// TwinCAT 3 PLC project Untitled1
// ProgramVersion: 3.1.4024.0
// libraries:
//   Tc2_Standard, * (Beckhoff Automation GmbH)
//   Tc2_System, * (Beckhoff Automation GmbH)
//   Tc3_Module, * (Beckhoff Automation GmbH)
// project tree:
//   / GlobalTextList.TcGTLO, PlcTask.TcTTO, Visualization Manager.TcVMO (not stored)
//   GVLs/ GIOL.TcGVL, Global_IO_assignment.TcPOU (not stored), GVL.TcGVL
//   POUs/ BINARY_TO_DEC.TcPOU, BLINK.TcPOU (not stored), MAIN.TcPOU, INMODE.TcPOU, Pulse.TcPOU, ROBOT_BIT_TRL.TcPOU
//   VISUs/ StandardPLCversenyVISU.TcVIS
// real-time tasks:
//   TASK PlcTask: cycle T#10ms, priority 20, ADS port 350
// I/O:
//   DEVICE Device 1 (EtherCAT), AmsNetId 5.86.98.224.2.1
//     Term 1 (EK1200) [EK1200-5000 EtherCAT Power supply (2A E-Bus)]
//       Term 2 (EL1008) [EL1008 8Ch. Dig. Input 24V, 3ms]
//       Term 3 (EL1008) [EL1008 8Ch. Dig. Input 24V, 3ms]
//       Term 4 (EL2008) [EL2008 8Ch. Dig. Output 24V, 0.5A]
//       Term 5 (EL2008) [EL2008 8Ch. Dig. Output 24V, 0.5A]
//       Term 6 (EL9011) [EL9011 End Terminal]
// variable links:
//   Untitled1/Untitled1 Instance <-> Device 1 (EtherCAT)/Term 1 (EK1200)/Term 2 (EL1008)
//     PlcTask Inputs/GIOL.xIn{0..7} <-> Channel {1..8}/Input  (8 links)
//   Untitled1/Untitled1 Instance <-> Device 1 (EtherCAT)/Term 1 (EK1200)/Term 3 (EL1008)
//     PlcTask Inputs/GIOL.xIn{8..15} <-> Channel {1..8}/Input  (8 links)
//   Untitled1/Untitled1 Instance <-> Device 1 (EtherCAT)/Term 1 (EK1200)/Term 4 (EL2008)
//     PlcTask Outputs/GIOL.Out{0..7} <-> Channel {1..8}/Output  (8 links)
//   Untitled1/Untitled1 Instance <-> Device 1 (EtherCAT)/Term 1 (EK1200)/Term 5 (EL2008)
//     PlcTask Outputs/GIOL.Out{8..15} <-> Channel {1..8}/Output  (8 links)

CONFIGURATION Untitled1
    RESOURCE PLC ON TwinCAT3
        TASK PlcTask(INTERVAL := T#10ms, PRIORITY := 20);
        PROGRAM MAIN WITH PlcTask : MAIN;
    END_RESOURCE
END_CONFIGURATION

// ---- GVLs/GIOL.TcGVL
{attribute 'qualified_only'}
VAR_GLOBAL
	xIn0 	AT%IX0.0:	BOOL;
	xIn1 	AT%IX0.1:	BOOL;
	xIn2 	AT%IX0.2:	BOOL;
	xIn3 	AT%IX0.3:	BOOL;
	xIn4 	AT%IX0.4:	BOOL;
	xIn5 	AT%IX0.5:	BOOL;
	xIn6 	AT%IX0.6:	BOOL;
	xIn7 	AT%IX0.7:	BOOL;
	
	xIn8 	AT%IX1.0:	BOOL;
	xIn9 	AT%IX1.1:	BOOL;
	xIn10 	AT%IX1.2:	BOOL;
	xIn11 	AT%IX1.3:	BOOL;
	xIn12 	AT%IX1.4:	BOOL;
	xIn13 	AT%IX1.5:	BOOL;
	xIn14 	AT%IX1.6:	BOOL;
	xIn15 	AT%IX1.7:	BOOL;
	
	Out0 	AT%QX0.0:	BOOL;
	Out1 	AT%QX0.1:	BOOL;
	Out2 	AT%QX0.2:	BOOL;
	Out3 	AT%QX0.3:	BOOL;
	Out4 	AT%QX0.4:	BOOL;
	Out5 	AT%QX0.5:	BOOL;
	Out6 	AT%QX0.6:	BOOL;
	Out7 	AT%QX0.7:	BOOL;
	
	
	Out8 	AT%QX1.0:	BOOL;
	Out9 	AT%QX1.1:	BOOL;
	Out10 	AT%QX1.2:	BOOL;
	Out11 	AT%QX1.3:	BOOL;
	Out12 	AT%QX1.4:	BOOL;
	Out13 	AT%QX1.5:	BOOL;
	Out14 	AT%QX1.6:	BOOL;
	Out15 	AT%QX1.7:	BOOL;
	
	In0 	:	BOOL;
	In1 	:	BOOL;
	In2 	:	BOOL;
	In3 	:	BOOL;
	In4 	:	BOOL;
	In5 	:	BOOL;
	In6 	:	BOOL;
	In7 	:	BOOL;
	
	In8 	:	BOOL;
	In9 	:	BOOL;
	In10 	:	BOOL;
	In11 	:	BOOL;
	In12 	:	BOOL;
	In13 	:	BOOL;
	In14 	:	BOOL;
	In15 	:	BOOL;
	
	bIn0 	:	BOOL;
	bIn1 	:	BOOL;
	bIn2 	:	BOOL;
	bIn3 	:	BOOL;
	bIn4 	:	BOOL;
	bIn5 	:	BOOL;
	bIn6 	:	BOOL;
	bIn7 	:	BOOL;
	
	bIn8 	:	BOOL;
	bIn9 	:	BOOL;
	bIn10 	:	BOOL;
	bIn11 	:	BOOL;
	bIn12 	:	BOOL;
	bIn13 	:	BOOL;
	bIn14 	:	BOOL;
	bIn15 	:	BOOL;
	
	TaskName : WSTRING := "Null Task";
	CaseNum  : INT := 0;
	
END_VAR

// ---- GVLs/GVL.TcGVL
{attribute 'qualified_only'}
VAR_GLOBAL
	In0 	:	BOOL;
	In1 	:	BOOL;
	In2 	:	BOOL;
	In3 	:	BOOL;
	In4 	:	BOOL;
	In5 	:	BOOL;
	In6 	:	BOOL;
	In7 	:	BOOL;
	
	In8 	:	BOOL;
	In9 	:	BOOL;
	In10 	:	BOOL;
	In11 	:	BOOL;
	In12 	:	BOOL;
	In13 	:	BOOL;
	In14 	:	BOOL;
	In15 	:	BOOL;
	
	TaskName : WSTRING := "Null Task";
	CaseNum  : INT := 0;
END_VAR

// ---- POUs/MAIN.TcPOU
PROGRAM MAIN
VAR
	INMODE : INMODE;
	
	CircularTablePosition1 : BOOL;
	CircularTablePosition2 : BOOL;
	CircularTablePosition3 : BOOL;
	PickupPointOccupied : BOOL; //NC gives back 1 when empty
	ManipulatorCircularEND : BOOL;
	ManipulatorFurnaceEND : BOOL;
	FurnaceIN : BOOL;
	FurnaceOUT : BOOL;
	FurnaceNotFULL : BOOL; //NC gives back 1 when empty
	CodeReader0 :  BOOL;
	CodeReader1 :  BOOL;
	StartButton : BOOL; //NO gives back 0 when not pressed
	SYSTEM_OK : BOOL;
	InConveyorOccupied : BOOL; //NO Gives back 0 when empty
	RobotIN_task_IN_Progress : BOOL;
	RobotOUT_task_IN_Progress : BOOL;
	
	CircTableRight : BOOL;
	CircTableLeft  : BOOL;
	PickupMotorGO : BOOL;
	SawMotor : BOOL;
	FurnaceGOin : BOOL;
	FurnaceGOout : BOOL;
	ManipulatorGOtoFurnace : BOOL;
	ManipulatorGOtoCircular : BOOL;
	FurnaceON : BOOL;
	ReaderTrigger : BOOL;
	ManipulatorVacuumON : BOOL; //monostabil
	ManipulatorZDOWN : BOOL; //monostabil!!!!!!
	FurnaceDoorUP :BOOL :=TRUE; //monostabil!!!!
 	RobotCOM0 : BOOL;
	RobotCOM1 : BOOL;
	CircularEJECT : BOOL; //monostabil!!!
	DelayTimer : TON;
	DelayAmount : TIME;
	DelayONtrigger : BOOL;
	FallTrig : F_TRIG;
	FallTrigCLK : BOOL;
	Pulse : Pulse;
	PulseSIGNAL : BOOL; 
	PulseTime : TIME;
	
	ScanCounter :INT := 0;
	FurnaceBurntime : TIME;
	
END_VAR

INMODE(); 
DelayTimer(IN:=DelayONtrigger,PT:=DelayAmount);
FallTrig(CLK:=FallTrigCLK);
Pulse(SIGNAL:=PulseSIGNAL,Pulse_time:=PulseTime);
CircularTablePosition1 := GIOL.In0;
CircularTablePosition2 := GIOL.In1;
CircularTablePosition3 := GIOL.In3;
PickupPointOccupied := GIOL.In2;
ManipulatorCircularEND := GIOL.In4;
ManipulatorFurnaceEND := GIOL.In7;
FurnaceIN := GIOL.In5;
FurnaceOUT := GIOL.In6;
FurnaceNotFULL := GIOL.In8;
CodeReader0 := GIOL.In9;
CodeReader1 := GIOL.In10;
StartButton := GIOL.In11;
SYSTEM_OK := GIOL.In12;
InConveyorOccupied := GIOL.In13;
RobotIN_task_IN_Progress := GIOL.In14;
RobotOUT_task_IN_Progress := GIOL.In15;

GIOL.Out0 := CircTableRight;
GIOL.Out1 := CircTableLeft;
GIOL.Out2 := PickupMotorGO;
GIOL.Out3 := SawMotor;
GIOL.Out4 := FurnaceGOin;
GIOL.Out5 := FurnaceGOout;
GIOL.Out6 := ManipulatorGOtoFurnace;
GIOL.Out7 := ManipulatorGOtoCircular;
GIOL.Out8 := FurnaceON;
GIOL.Out9 := ReaderTrigger;
GIOL.Out10 := ManipulatorVacuumON;
GIOL.Out11 := ManipulatorZDOWN;
GIOL.Out12 := FurnaceDoorUP;
GIOL.Out13 := RobotCOM0;
GIOL.Out14 := RobotCOM1;
GIOL.Out15 := CircularEJECT;

IF SYSTEM_OK THEN
CASE GIOL.CaseNum OF
	
	0:GIOL.TaskName:="Idle position, wait for start button";
		IF StartButton THEN
			GIOL.CaseNum:=10;
		END_IF
		
	10:GIOL.TaskName:="Check for workpiece on inconveyor";
		IF InConveyorOccupied AND FurnaceNotFULL THEN
			DelayAmount := T#1S;
			GIOL.CaseNum := 20;
		ELSE 
			GIOL.CaseNum:=0;
		END_IF
		
	20:GIOL.TaskName:="Wait for 1 sec";
		DelayONtrigger := TRUE;
		IF DelayTimer.Q THEN
			DelayONtrigger := FALSE;
			GIOL.CaseNum:=30;
		END_IF
		
	30:GIOL.TaskName:="Open furnace if in";
		IF FurnaceOUT THEN
			GIOL.CaseNum := 40;
		ELSE
			FurnaceGOout := TRUE;
			FurnaceGOin :=FALSE;
			DelayAmount := T#4S;
			GIOL.CaseNum := 35;
		END_IF
		
	35:GIOL.TaskName:="Open Furnace";
		DelayONtrigger := TRUE;
		IF DelayTimer.Q THEN
			GIOL.CaseNum := 40;
			DelayONtrigger := FALSE;
			FurnaceGOin := FALSE;
		END_IF
		
	40:GIOL.TaskName:="Give Robot load command";
		RobotCOM0 := 0;
		RobotCOM1 := 1;
		GIOL.CaseNum := 50;
		
	50:GIOL.TaskName:="Load workpiece into furnace";
		FallTrigCLK := RobotIN_task_IN_Progress;
		IF RobotIN_task_IN_Progress THEN
			RobotCOM0 := 0;
			RobotCOM1 := 0;
		END_IF
		IF FallTrig.Q THEN
			GIOL.CaseNum := 60;
		END_IF
		
	60:GIOL.TaskName:="Identify workpiece";
		IF NOT FurnaceNotFULL THEN
			ReaderTrigger := TRUE;
			PulseTime:=T#400MS;
			PulseSIGNAL:=TRUE;
			GIOL.CaseNum:=61;
		END_IF
	
	61:GIOL.TaskName:="Identify workpiece";
		IF NOT PulseSIGNAL THEN
			PulseTime:=T#2S;
			PulseSIGNAL:=TRUE;
			GIOL.CaseNum := 62;
			ReaderTrigger:=FALSE;
		END_IF
		
	62:GIOL.TaskName:="Identify workpiece";
		IF NOT PulseSIGNAL AND NOT CodeReader0 AND NOT CodeReader1 THEN
			ScanCounter := ScanCounter + 1;
			GIOL.CaseNum:=60;
			IF ScanCounter = 2 THEN
				GIOL.CaseNum:=0;
				ScanCounter:=0;
			END_IF
		END_IF
		
		IF NOT CodeReader0 AND CodeReader1 THEN
			FurnaceBurntime := T#5000MS;
			GIOL.CaseNum := 70;
		END_IF
		IF CodeReader0 AND NOT CodeReader1 THEN
			FurnaceBurntime := T#1500MS;
			GIOL.CaseNum := 70;
		END_IF
		IF CodeReader0 AND CodeReader1 THEN
			FurnaceBurntime := T#3000MS;
			GIOL.CaseNum := 70;
		END_IF
	
	70:GIOL.TaskName:="Pull workpiece into furnace";
		FurnaceGOin:=TRUE;
		FurnaceGOout:=FALSE;	
		GIOL.CaseNum:=71;
		ScanCounter:=0;
		
	71:GIOL.TaskName:="Pull workpiece into furnace";
		IF FurnaceIN THEN
			FurnaceGOin:=FALSE;
			FurnaceGOout:=FALSE;
			FurnaceDoorUP:=FALSE;
			DelayAmount:=T#1S;
			GIOL.CaseNum:=72;
		END_IF
	72:GIOL.TaskName:="Close furnace door";
		DelayONtrigger:=TRUE;
		IF DelayTimer.Q THEN
			DelayONtrigger:=FALSE;
			GIOL.CaseNum:=73;
			FurnaceON:=TRUE;
			DelayAmount:=FurnaceBurntime;
		END_IF
	73:GIOL.TaskName:="BURN!!!!";
		DelayONtrigger:=TRUE;
		IF DelayTimer.Q THEN
			DelayONtrigger:=FALSE;
			FurnaceON:=FALSE;
			FurnaceDoorUP:=TRUE;
			DelayAmount:=T#1S;
			GIOL.CaseNum:=80;
		END_IF
		
	80:GIOL.TaskName:="Open furnace door";
		DelayONtrigger:=TRUE;
		IF DelayTimer.Q THEN
			DelayONtrigger:=FALSE;
			FurnaceGOout:=TRUE;
			FurnaceGOin:=FALSE;
			GIOL.CaseNum:=90;
		END_IF
		
	90:GIOL.TaskName:="Send out workpiece";
		IF FurnaceOUT THEN
			ManipulatorGOtoFurnace:=TRUE;
			ManipulatorGOtoCircular:=FALSE;
			IF CircularTablePosition1 THEN
				GIOL.CaseNum:=100;
			ELSE
				GIOL.CaseNum:=91;
				CircTableLeft:=TRUE;
			END_IF			
		END_IF
		
	91:GIOL.TaskName:="Adjust circular table";
		IF CircularTablePosition1 THEN
			CircTableLeft := FALSE;
			GIOL.CaseNum  := 100;
		END_IF
		
	100:GIOL.TaskName:="Take workpiece to table";
		IF ManipulatorFurnaceEND THEN
			ManipulatorGOtoFurnace:=FALSE;
			ManipulatorGOtoCircular:=FALSE;
			ManipulatorZDOWN:=TRUE;
			ManipulatorVacuumON:=TRUE;
			DelayAmount:=T#1S;
			GIOL.CaseNum:=101;
		END_IF
		
	101:GIOL.TaskName:="Take workpiece to table";
		DelayONtrigger:=TRUE;
		IF DelayTimer.Q THEN
			DelayONtrigger:=FALSE;
			ManipulatorZDOWN:=FALSE;
			DelayAmount := T#500MS;
			GIOL.CaseNum:=102;
		END_IF
		
	102:GIOL.TaskName:="Take workpiece to table";
		DelayONtrigger:=TRUE;
		IF DelayTimer.Q THEN
			DelayONtrigger:=FALSE;
			ManipulatorGOtoCircular:=TRUE;
			GIOL.CaseNum:=103;
		END_IF
		
	103:GIOL.TaskName:="Take workpiece to table";
		IF ManipulatorCircularEND THEN
			ManipulatorZDOWN:=TRUE;
			DelayAmount:=T#500MS;
			GIOL.CaseNum:=104;
		END_IF
		
	104:GIOL.TaskName:="Take workpiece to table";
		DelayONtrigger:=TRUE;
		IF DelayTimer.Q THEN
			DelayONtrigger:=FALSE;
			ManipulatorVacuumON:=FALSE;
			ManipulatorZDOWN:=FALSE;
			DelayAmount:=T#500MS;
			GIOL.CaseNum:=105;
		END_IF
		
	105:GIOL.TaskName:="Wait for putdown";
		DelayONtrigger:=TRUE;
		IF DelayTimer.Q THEN
			CircTableRight:=TRUE;
			DelayONtrigger:=FALSE;
			GIOL.CaseNum:=110;
		END_IF
		
		
	110:GIOL.TaskName:="SAW Operation";
		IF CircularTablePosition3 THEN
			CircTableRight:=FALSE;
			SawMotor:=TRUE;
			DelayAmount:=T#2S;
			GIOL.CaseNum:=111;
		END_IF
	
	111:GIOL.TaskName:="SAW Operation";
		DelayONtrigger:=TRUE;
		IF DelayTimer.Q THEN
			DelayONtrigger:=FALSE;
			SawMotor:=FALSE;
			CircTableRight:=TRUE;
			GIOL.CaseNum:=120;
		END_IF
		
	120:GIOL.TaskName:="SAW Operation";
		IF CircularTablePosition2 THEN
			CircTableRight:=FALSE;
			DelayAmount:=T#500MS;
			GIOL.CaseNum:=130;
		END_IF
		
	130:GIOL.TaskName:="Eject workpiece from table";
		DelayONtrigger:=TRUE;
		IF DelayTimer.Q THEN
			DelayONtrigger:=FALSE;
			CircularEJECT:=TRUE;
			DelayAmount:=T#1000MS;
			GIOL.CaseNum:=131;
		END_IF
		
	131:GIOL.TaskName:="Eject workpiece from table";
		DelayONtrigger:=TRUE;
		IF DelayTimer.Q THEN
			DelayONtrigger:=FALSE;
			CircularEJECT:=FALSE;
			PickupMotorGO:=TRUE;
			CircTableLeft:=TRUE;
			GIOL.CaseNum:=140;
		END_IF
		
	140:GIOL.TaskName:="Take workpiece to pickup point";
		IF NOT PickupPointOccupied THEN
			PickupMotorGO:=FALSE;
		END_IF
		IF CircularTablePosition1 THEN 
			CircTableLeft:=FALSE;
			RobotCOM0:=1;
			RobotCOM1:=1;
			GIOL.CaseNum:=150;
		END_IF
			
	150:GIOL.TaskName:="Take workpiece to endpoint";
		FallTrigCLK :=  RobotOUT_task_IN_Progress;
		IF RobotOUT_task_IN_Progress THEN
			RobotCOM0 := 0;
			RobotCOM1 := 0;
		END_IF
		IF FallTrig.Q THEN
			GIOL.CaseNum := 160;
		END_IF
		
	160:GIOL.TaskName:="Finished task";
		GIOL.CaseNum:=10;
	
	ELSE
		GIOL.CaseNum:=0;
END_CASE
ELSE
	GIOL.CaseNum := 0;
	CircTableRight := 0;
	CircTableLeft := 0;
	PickupMotorGO := 0;
	SawMotor := 0;
	FurnaceGOin := 0;
	FurnaceGOout := 0;
	ManipulatorGOtoFurnace := 0;
	ManipulatorGOtoCircular := 0;
	RobotCOM0 := 0;
	RobotCOM1 :=0;
	FurnaceON := 0;
	ReaderTrigger := 0;
	ManipulatorVacuumON := 0;
	ManipulatorZDOWN := 0;
	CircularEJECT := 0;
END_IF
//some random change

END_PROGRAM

// ---- POUs/INMODE.TcPOU
FUNCTION_BLOCK INMODE
VAR_INPUT
	INState : BOOL :=  FALSE;
END_VAR

IF INState THEN
	GIOL.In0 := GIOL.bIn0;
	GIOL.In1 := GIOL.bIn1;
	GIOL.In2 := GIOL.bIn2;
	GIOL.In3 := GIOL.bIn3;
	GIOL.In4 := GIOL.bIn4;
	GIOL.In5 := GIOL.bIn5;
	GIOL.In6 := GIOL.bIn6;
	GIOL.In7 := GIOL.bIn7;
	
	GIOL.In8 := GIOL.bIn8;
	GIOL.In9 := GIOL.bIn9;
	GIOL.In10 := GIOL.bIn10;
	GIOL.In11 := GIOL.bIn11;
	GIOL.In12 := GIOL.bIn12;
	GIOL.In13 := GIOL.bIn13;
	GIOL.In14 := GIOL.bIn14;
	GIOL.In15 := GIOL.bIn15;
ELSE
	GIOL.In0 := GIOL.xIn0;
	GIOL.In1 := GIOL.xIn1;
	GIOL.In2 := GIOL.xIn2;
	GIOL.In3 := GIOL.xIn3;
	GIOL.In4 := GIOL.xIn4;
	GIOL.In5 := GIOL.xIn5;
	GIOL.In6 := GIOL.xIn6;
	GIOL.In7 := GIOL.xIn7;
	
	GIOL.In8 := GIOL.xIn8;
	GIOL.In9 := GIOL.xIn9;
	GIOL.In10 := GIOL.xIn10;
	GIOL.In11 := GIOL.xIn11;
	GIOL.In12 := GIOL.xIn12;
	GIOL.In13 := GIOL.xIn13;
	GIOL.In14 := GIOL.xIn14;
	GIOL.In15 := GIOL.xIn15;
END_IF

END_FUNCTION_BLOCK

// ---- POUs/Pulse.TcPOU
FUNCTION_BLOCK Pulse
VAR_INPUT
	Pulse_time : TIME; // Az impulzus ideje, ennyi idő után kapcsol le
END_VAR
VAR_OUTPUT
	
END_VAR

VAR
clk :TON;

END_VAR
VAR_IN_OUT
	SIGNAL  : BOOL; // A jel amit kapcsolni kell
END_VAR

clk(IN:=SIGNAL,PT:=Pulse_time);

IF clk.Q THEN
	SIGNAL := FALSE;
		
END_IF

END_FUNCTION_BLOCK

// ---- POUs/BINARY_TO_DEC.TcPOU
FUNCTION_BLOCK BINARY_TO_DEC
VAR_INPUT
	BIN0 : BOOL; //Bemenet MSB
	BIN1 : BOOL; //Bemenet
	BIN2 : BOOL; //Bemenet 
END_VAR
VAR_OUTPUT
	ID : INT; // kimeneti int
	
END_VAR
VAR
	bH : ARRAY [0..2] OF  INT; // helyiértékek értékei
	i : UINT;
END_VAR


FOR i :=0 TO 2 DO
	bH[i] :=(LREAL_TO_INT( EXPT(2,i)));
	
END_FOR
ID := (BOOL_TO_INT(BIN0)* bH[0])+ BOOL_TO_INT(BIN1)*bH[1]+BOOL_TO_INT(BIN2)*bH[2];

END_FUNCTION_BLOCK

// ---- POUs/ROBOT_BIT_TRL.TcPOU
FUNCTION_BLOCK ROBOT_BIT_TRL
VAR_INPUT
	ROBPOZ : INT; // Robot pozíció száma
	
END_VAR

VAR_OUTPUT
	POZ0 :BOOL; //Kimenet bit MSB
	POZ1 :BOOL; //Kimenet
	
	
END_VAR
VAR
	
END_VAR

CASE ROBPOZ OF
0:
POZ0 := 0;
POZ1 := 0;


1:
POZ0 := 1;
POZ1 :=0;


2:
POZ0 :=0;
POZ1 :=1;

3:
POZ0 :=1;
POZ1 :=1;

END_CASE

END_FUNCTION_BLOCK

// ---- GlobalTextList.TcGTLO
TEXTLIST GlobalTextList
  216 = 'CASE: %d'
  404 = 'EXECUTING: %s'
  848 = 'IN 0'
  11 = 'IN 1'
  929 = 'INPUT MODE'
  620 = 'OUT 0'
  877 = 'OUT 1'
END_TEXTLIST

// ---- VISUs/StandardPLCversenyVISU.TcVIS
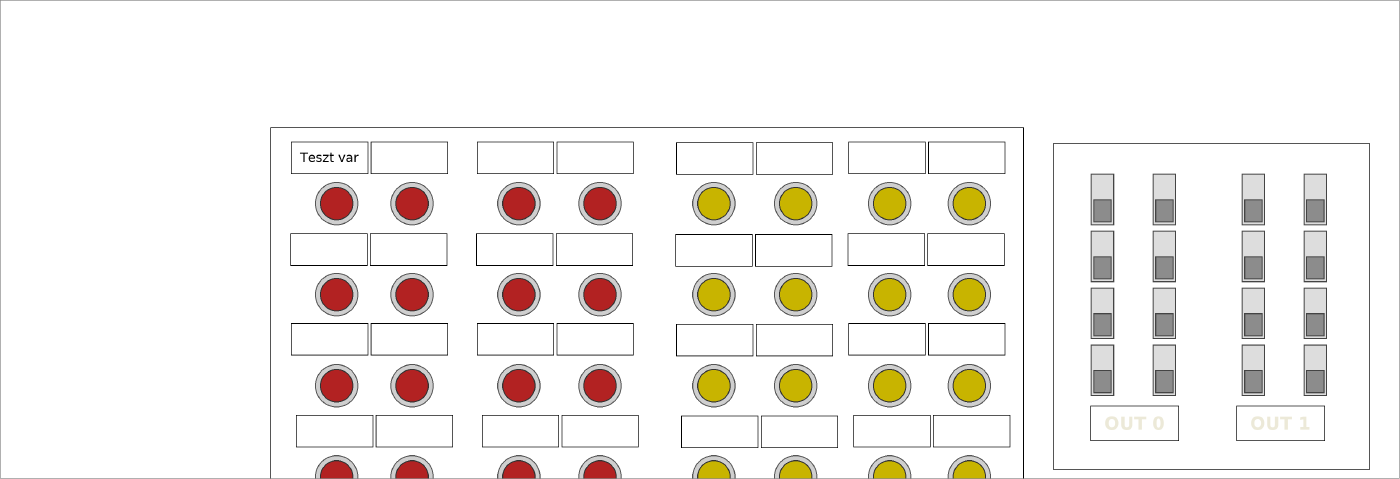
VISUALIZATION StandardPLCversenyVISU  // 1967x673
    Rectangle (1769,708 331x259)
    Rectangle (1480,201 444x459)
    Rectangle (380,179 1058x846)
    Lamp1 (438,251 70x70), variable: GIOL.out0, style: Lamp-Lamp1-Red
    Lamp1 (544,251 70x70), variable: GIOL.out1, style: Lamp-Lamp1-Red
    Lamp1 (694,251 70x70), variable: GIOL.out8, style: Lamp-Lamp1-Red
    Lamp1 (808,251 70x70), variable: GIOL.out9, style: Lamp-Lamp1-Red
    Lamp1 (438,379 70x70), variable: GIOL.out2, style: Lamp-Lamp1-Red
    Lamp1 (544,379 70x70), variable: GIOL.out3, style: Lamp-Lamp1-Red
    Lamp1 (694,379 70x70), variable: GIOL.out10, style: Lamp-Lamp1-Red
    Lamp1 (808,379 70x70), variable: GIOL.out11, style: Lamp-Lamp1-Red
    Lamp1 (438,507 70x70), variable: GIOL.out4, style: Lamp-Lamp1-Red
    Lamp1 (544,507 70x70), variable: GIOL.out5, style: Lamp-Lamp1-Red
    Lamp1 (694,507 70x70), variable: GIOL.out12, style: Lamp-Lamp1-Red
    Lamp1 (808,507 70x70), variable: GIOL.out13, style: Lamp-Lamp1-Red
    Lamp1 (438,635 70x70), variable: GIOL.out6, style: Lamp-Lamp1-Red
    Lamp1 (544,635 70x70), variable: GIOL.out7, style: Lamp-Lamp1-Red
    Lamp1 (694,635 70x70), variable: GIOL.out14, style: Lamp-Lamp1-Red
    Lamp1 (808,635 70x70), variable: GIOL.out15, style: Lamp-Lamp1-Red
    Lamp1 (968,251 70x70), variable: GIOL.in0, style: Lamp-Lamp1-Yellow
    Lamp1 (1083,251 70x70), variable: GIOL.in1, style: Lamp-Lamp1-Yellow
    Lamp1 (1215,251 70x70), variable: GIOL.in8, style: Lamp-Lamp1-Yellow
    Lamp1 (1327,251 70x70), variable: GIOL.in9, style: Lamp-Lamp1-Yellow
    Lamp1 (968,379 70x70), variable: GIOL.in2, style: Lamp-Lamp1-Yellow
    Lamp1 (1083,379 70x70), variable: GIOL.in3, style: Lamp-Lamp1-Yellow
    Lamp1 (1215,379 70x70), variable: GIOL.in10, style: Lamp-Lamp1-Yellow
    Lamp1 (1327,379 70x70), variable: GIOL.in11, style: Lamp-Lamp1-Yellow
    Lamp1 (968,507 70x70), variable: GIOL.in4, style: Lamp-Lamp1-Yellow
    Lamp1 (1083,507 70x70), variable: GIOL.in5, style: Lamp-Lamp1-Yellow
    Lamp1 (1215,507 70x70), variable: GIOL.in12, style: Lamp-Lamp1-Yellow
    Lamp1 (1327,507 70x70), variable: GIOL.in13, style: Lamp-Lamp1-Yellow
    Lamp1 (968,635 70x70), variable: GIOL.in6, style: Lamp-Lamp1-Yellow
    Lamp1 (1083,635 70x70), variable: GIOL.in7, style: Lamp-Lamp1-Yellow
    Lamp1 (1215,635 70x70), variable: GIOL.in14, style: Lamp-Lamp1-Yellow
    Lamp1 (1327,635 70x70), variable: GIOL.in15, style: Lamp-Lamp1-Yellow
    Rectangle (700,733 124x49), "OUT 1"
    Rectangle (988,728 124x49), "IN 0"
    Rectangle (450,733 124x49), "OUT 0"
    Rectangle (1229,726 124x49), "IN 1"
    Rectangle (505,888 695x68), "EXECUTING: %s", text variable: GIOL.TaskName
    DipSwitch (1600,240 72x80), variable: GIOL.out1, behaviour: TOGGLE, style: Switch-DipSwitch-Gray
    DipSwitch (1513,240 72x80), variable: GIOL.out0, behaviour: TOGGLE, style: Switch-DipSwitch-Gray
    DipSwitch (1600,320 72x80), variable: GIOL.out3, behaviour: TOGGLE, style: Switch-DipSwitch-Gray
    DipSwitch (1513,320 72x80), variable: GIOL.out2, behaviour: TOGGLE, style: Switch-DipSwitch-Gray
    DipSwitch (1600,400 72x80), variable: GIOL.out5, behaviour: TOGGLE, style: Switch-DipSwitch-Gray
    DipSwitch (1513,400 72x80), variable: GIOL.out4, behaviour: TOGGLE, style: Switch-DipSwitch-Gray
    DipSwitch (1600,480 72x80), variable: GIOL.out7, behaviour: TOGGLE, style: Switch-DipSwitch-Gray
    DipSwitch (1513,480 72x80), variable: GIOL.out6, behaviour: TOGGLE, style: Switch-DipSwitch-Gray
    DipSwitch (1812,240 72x80), variable: GIOL.out9, behaviour: TOGGLE, style: Switch-DipSwitch-Gray
    DipSwitch (1725,240 72x80), variable: GIOL.out8, behaviour: TOGGLE, style: Switch-DipSwitch-Gray
    DipSwitch (1812,320 72x80), variable: GIOL.out11, behaviour: TOGGLE, style: Switch-DipSwitch-Gray
    DipSwitch (1725,320 72x80), variable: GIOL.out10, behaviour: TOGGLE, style: Switch-DipSwitch-Gray
    DipSwitch (1812,400 72x80), variable: GIOL.out13, behaviour: TOGGLE, style: Switch-DipSwitch-Gray
    DipSwitch (1725,400 72x80), variable: GIOL.out12, behaviour: TOGGLE, style: Switch-DipSwitch-Gray
    DipSwitch (1812,480 72x80), variable: GIOL.out15, behaviour: TOGGLE, style: Switch-DipSwitch-Gray
    DipSwitch (1725,480 72x80), variable: GIOL.out14, behaviour: TOGGLE, style: Switch-DipSwitch-Gray
    Rectangle (1737,570 124x49), "OUT 1"
    Rectangle (1532,570 124x49), "OUT 0"
    Rectangle (1970,201 444x459)
    DipSwitch (2093,240 72x80), variable: GIOL.bIn1, behaviour: TOGGLE, style: Switch-DipSwitch-Gray
    DipSwitch (2006,240 72x80), variable: GIOL.bIn0, behaviour: TOGGLE, style: Switch-DipSwitch-Gray
    DipSwitch (2093,320 72x80), variable: GIOL.bIn3, behaviour: TOGGLE, style: Switch-DipSwitch-Gray
    DipSwitch (2006,320 72x80), variable: GIOL.bIn2, behaviour: TOGGLE, style: Switch-DipSwitch-Gray
    DipSwitch (2093,400 72x80), variable: GIOL.bIn5, behaviour: TOGGLE, style: Switch-DipSwitch-Gray
    DipSwitch (2006,400 72x80), variable: GIOL.bIn4, behaviour: TOGGLE, style: Switch-DipSwitch-Gray
    DipSwitch (2093,480 72x80), variable: GIOL.bIn7, behaviour: TOGGLE, style: Switch-DipSwitch-Gray
    DipSwitch (2006,480 72x80), variable: GIOL.bIn6, behaviour: TOGGLE, style: Switch-DipSwitch-Gray
    DipSwitch (2305,240 72x80), variable: GIOL.bIn9, behaviour: TOGGLE, style: Switch-DipSwitch-Gray
    DipSwitch (2218,240 72x80), variable: GIOL.bIn8, behaviour: TOGGLE, style: Switch-DipSwitch-Gray
    DipSwitch (2305,320 72x80), variable: GIOL.bIn11, behaviour: TOGGLE, style: Switch-DipSwitch-Gray
    DipSwitch (2218,320 72x80), variable: GIOL.bIn10, behaviour: TOGGLE, style: Switch-DipSwitch-Gray
    DipSwitch (2305,400 72x80), variable: GIOL.bIn13, behaviour: TOGGLE, style: Switch-DipSwitch-Gray
    DipSwitch (2218,400 72x80), variable: GIOL.bIn12, behaviour: TOGGLE, style: Switch-DipSwitch-Gray
    DipSwitch (2305,480 72x80), variable: GIOL.bIn15, behaviour: TOGGLE, style: Switch-DipSwitch-Gray
    DipSwitch (2218,480 72x80), variable: GIOL.bIn14, behaviour: TOGGLE, style: Switch-DipSwitch-Gray
    Rectangle (2230,570 124x49), "IN 1"
    Rectangle (2025,570 124x49), "IN 0"
    Rectangle (1210,888 153x68), "CASE: %d", text variable: GIOL.CaseNum
    DipSwitch (1818,753 116x113), variable: MAIN.INMODE.INState, behaviour: TOGGLE, style: Switch-DipSwitch-Gray
    Rectangle (1828,898 226x49), "INPUT MODE"
    Lamp1 (1963,775 70x70), variable: MAIN.INMODE.INState, style: Lamp-Lamp1-Yellow
    Rectangle (409,199 108x45), "Teszt var"
    Rectangle (521,199 108x45)
    Rectangle (670,199 108x45)
    Rectangle (782,199 108x45)
    Rectangle (950,200 108x45)
    Rectangle (1062,200 108x45)
    Rectangle (1192,199 108x45)
    Rectangle (1304,199 108x45)
    Rectangle (408,328 108x45)
    Rectangle (520,328 108x45)
    Rectangle (669,328 108x45)
    Rectangle (781,328 108x45)
    Rectangle (949,329 108x45)
    Rectangle (1061,329 108x45)
    Rectangle (1191,328 108x45)
    Rectangle (1303,328 108x45)
    Rectangle (409,454 108x45)
    Rectangle (521,454 108x45)
    Rectangle (670,454 108x45)
    Rectangle (782,454 108x45)
    Rectangle (950,455 108x45)
    Rectangle (1062,455 108x45)
    Rectangle (1192,454 108x45)
    Rectangle (1304,454 108x45)
    Rectangle (416,583 108x45)
    Rectangle (528,583 108x45)
    Rectangle (677,583 108x45)
    Rectangle (789,583 108x45)
    Rectangle (957,584 108x45)
    Rectangle (1069,584 108x45)
    Rectangle (1199,583 108x45)
    Rectangle (1311,583 108x45)
END_VISUALIZATION
